// TIA Portal V20 export
FUNCTION "FC_CheckTimeout" : Void   // FC34, SCL
{ S7_Optimized_Access := 'TRUE' }
// stored: SetENOAutomatically false
   VAR_INPUT
      iCondition : Bool;
      iTime : Time;
   END_VAR
   VAR_OUTPUT
      oTimeoutOccurred : Bool;
   END_VAR
   VAR_IN_OUT
      ioTimer : TON_TIME;
   END_VAR
BEGIN
   REGION Description header 
       //==================================================================================
       // POSALUX Swiss SA / (C) Copyright 2025
       //----------------------------------------------------------------------------------
       // Title: CheckTimeout
       // Comment/Function: Start a Timeout control according conditions
       //                   Set a bit at the end of the timer
       // Author: Fabien WALDT
       // Engineering: TIA Portal v17
       //----------------------------------------------------------------------------------
       // Change log table:
       // Version  | Date     | Expert in charge | Changes applied
       // ---------|----------|------------------|-----------------------------------------
       // 00.00.01 | 20250423 | WFA              | First released version
       // =================================================================================
   END_REGION
   // Configuration du timer
   #ioTimer.PT := #iTime;

   // Activation du timer si la condition est vraie
   #ioTimer.IN := #iCondition;

   // Vérification du timeout
   IF #ioTimer.Q THEN
       #oTimeoutOccurred := true;
   ELSIF "MCP1_In".reset THEN
       #oTimeoutOccurred := false;
   END_IF;
END_FUNCTION
